Yaskawa INFORM job: 1-X.JBI

/JOB
//NAME 1-X
///FOLDERNAME INNE
//POS
///NPOS 2,2,0,0,0,0
///TOOL 0
///POSTYPE PULSE
///PULSE
C00000=1484,21688,49925,260,89810,865
C00001=237611,-89580,-19083,2248,32818,80213
BC00000=55035,1064966,688932
BC00001=311297,1064968,688937
//INST
///DATE 2023/11/08 10:34
///ATTR SC,RW
///GROUP1 RB1,BS1
NOP
MOVJ C00000 BC00000 VJ=0.78
MOVJ C00001 BC00001 VJ=0.78
SFTOF
END
